INTERFACE itfStatusFlags

PROPERTY pBuffering : BOOL
GET
END_GET
SET
END_SET
END_PROPERTY

PROPERTY pDosing : BOOL
GET
END_GET
SET
END_SET
END_PROPERTY

PROPERTY pFault : BOOL
GET
END_GET
SET
END_SET
END_PROPERTY

PROPERTY pHaltBatch : BOOL
GET
END_GET
SET
END_SET
END_PROPERTY

PROPERTY pLowProduct : BOOL
GET
END_GET
SET
END_SET
END_PROPERTY

PROPERTY pMixing : BOOL
GET
END_GET
SET
END_SET
END_PROPERTY

PROPERTY pStoring : BOOL
GET
END_GET
SET
END_SET
END_PROPERTY

END_INTERFACE

(* stored: Version 1.1.0.1, ProductVersion 3.1.4024.12
   Itf itfStatusFlags: Id {5400ab44-ec83-4c4b-85ed-9950e264603c}
   Property pBuffering: Id {60a04fab-75d3-4bc3-a2f0-51ddbdc8b959}
   Get Get: Id {34e3a455-f104-4a4e-8a2a-db35c0761a9a}
   Set Set: Id {bdbf4bd5-a1b7-4f24-8cd2-430b2e7c679d}
   Property pDosing: Id {3174992c-cecc-492d-abc3-b4b3b5bd448d}
   Get Get: Id {4841e78a-ea72-49aa-88d5-eb871677be7b}
   Set Set: Id {c7d29b9f-f7d7-4918-b774-9aff2cf74d84}
   Property pFault: Id {1c04828f-8294-45c5-9d5e-dc58853156bd}
   Get Get: Id {b6309bd3-f155-429b-b90b-f446d9c744be}
   Set Set: Id {b7dda360-9fe0-477e-8428-184df8c8989f}
   Property pHaltBatch: Id {6a0e6a06-6288-47c2-ae87-fb91283eb286}
   Get Get: Id {20eb6b27-52bb-458b-b248-7ed115a8d69e}
   Set Set: Id {88282263-693d-4131-a09c-312d5ef4a479}
   Property pLowProduct: Id {ae3377fa-d71a-4c09-ab8c-999fbdc66a51}
   Get Get: Id {b6c12e94-7b20-4366-bb73-ff05db81e7c2}
   Set Set: Id {b3de28e5-accc-4a7b-8f0d-24070e1091eb}
   Property pMixing: Id {1c7d3f8a-656d-47ed-8c6c-8d412d104db6}
   Get Get: Id {2f852e38-7399-4594-a53c-4641dd7f0aa8}
   Set Set: Id {a4e9ec5f-8b5d-4c66-9d8c-43a4fa47bdc0}
   Property pStoring: Id {8485a48b-b19a-4727-87e0-e8dfbf54f1ad}
   Get Get: Id {fa9b4529-9ef7-43b0-a7eb-88f1e3e4c35e}
   Set Set: Id {61630e9c-6cb1-4054-afda-c477b47975ef} *)
